// TIA Portal project "AWL LIBRO 1" (V11)

(* hardware
DEVICE "S7300/ET200 station_1"  SIMATIC 300-Station
   slot 0: "Perfil soporte_0"  Rail  6ES7 390-1***0-0AA0
   slot 2: "PLC_1"  CPU 313C-2 DP  6ES7 313-6CF03-0AB0  V2.6
      slot 0: "Interfaz MPI_1"  MPI
      slot 1: "Interfaz DP_1"  DP
      slot 2: "DI16/DO16_1"  DI16/DO16
      slot 4: "Contaje_1"  Counter
*)

// ===== PLC "PLC_1"  CPU 313C-2 DP =====

VAR_GLOBAL   // PLC tag table "Tabla de variables estándar"
   "MARCHA" AT %E0.0 : Bool;
   "PARO" AT %E0.1 : Bool;
   "RELE TERMICO" AT %E0.2 : Bool;
   "MOTOR" AT %A0.0 : Bool;
   "LED MARCHA" AT %A0.1 : Bool;
   "LED DESCARGA" AT %A0.2 : Bool;
   "LED PARO" AT %A0.3 : Bool;
   "LED AVERIA" AT %A0.4 : Bool;
   "SALIDAS" AT %AB0 : Byte;
   "Tag_1" AT %T0 : Timer;
   "Tag_2" AT %M10.0 : Bool;
   "Tag_3" AT %M10.1 : Bool;
   "Tag_4" AT %MB0 : Byte;
   "Tag_5" AT %M10.2 : Bool;
END_VAR

ORGANIZATION_BLOCK "Main"   // OB1, STL
TITLE = "Main Program Sweep (Cycle)"
{ S7_Optimized_Access := 'FALSE' }
VERSION : 0.1
   VAR_TEMP
      OB1_EV_CLASS : Byte;   // Bits 0-3 = 1 (Coming event), Bits 4-7 = 1 (Event class 1)
      OB1_SCAN_1 : Byte;   // 1 (Cold restart scan 1 of OB 1), 3 (Scan 2-n of OB 1)
      OB1_PRIORITY : Byte;   // Priority of OB Execution
      OB1_OB_NUMBR : Byte;   // 1 (Organization block 1, OB1)
      OB1_RESERVED_1 : Byte;   // Reserved for system
      OB1_RESERVED_2 : Byte;   // Reserved for system
      OB1_PREV_CYCLE : Int;   // Cycle time of previous OB1 scan (milliseconds)
      OB1_MIN_CYCLE : Int;   // Minimum cycle time of OB1 (milliseconds)
      OB1_MAX_CYCLE : Int;   // Maximum cycle time of OB1 (milliseconds)
      OB1_DATE_TIME : Date_And_Time;   // Date and time OB1 started
   END_VAR
BEGIN

REGION Network 1: EJERCICIO 1 LIBRO
         AN    "Tag_2";  // REPOSO LED PARO ENCENDIDA.
         FP    "Tag_3";
         JNB   _004;
         L     B#16#8;
         T     "SALIDAS";
   _004: NOP   0;

         A     "MARCHA";
         JNB   _001;
         L     B#16#03;  // ARRANCA MOTOR Y LED MARCHA.
         T     "SALIDAS";
   _001: NOP   0;
         A     "PARO";
         A     "MOTOR";
         JNB   _002;
         L     B#16#05;  // ENTRA EN DESCARGA DURANTE 4S.
         T     "SALIDAS";
   _002: NOP   0;
         A     "LED DESCARGA";
         L     S5T#4S;  // TEMPORIZDO DESCARGA 4S.
         SD    "Tag_1";
         A     "Tag_1";
         JNB   _003;
         L     B#16#8;  // SE PARA Y ENCIENDE LED PARO.
         T     "SALIDAS";
   _003: NOP   0;
         A     "RELE TERMICO";  // DISPARO TERMICO.
         A     "MOTOR";
         JNB   _005;
         L     B#16#18;
         T     "SALIDAS";
   _005: NOP   0;
         A     "RELE TERMICO";
         FN    "Tag_5";
         JNB   _006;
         L     B#16#8;
         T     "SALIDAS";
   _006: NOP   0;
END_REGION
END_ORGANIZATION_BLOCK